// TIA Portal V17 export
// export: Created 2024-09-03T21:54:53.6894655Z, ExportSetting WithDefaults, DisplayName Totally Integrated Automation Portal, DisplayVersion V17 Update 7, DisplayName TIA Portal Openness, DisplayVersion V17 Update 7, DisplayName TIA Portal Version Control Interface, DisplayVersion V17, DisplayName SINAMICS Startdrive Advanced, DisplayVersion V17 SP2, DisplayName SINAMICS Startdrive G110M, G120, G120C, G120D, G120P, G115D, DisplayVersion V17 SP2, DisplayName SINAMICS Startdrive G130, G150, S120, S150, SINAMICS MV, S210, DisplayVersion V17 SP2, DisplayName STEP 7 Professional, DisplayVersion V17 Update 7, DisplayName STEP 7 Safety, DisplayVersion V17 Update 6, DisplayName WinCC Advanced / Unified PC, DisplayVersion V17 Update 7
ORGANIZATION_BLOCK "Startup"   // OB124, LAD, Startup
TITLE = "Complete Restart"
{ S7_Optimized_Access := 'TRUE' }
VERSION : 0.1
// stored: AutoNumber true, IsIECCheckEnabled false, SetENOAutomatically false
   VAR_INPUT
      LostRetentive : Bool;   // True if retentive data are lost
      LostRTC : Bool;   // True if date and time are lost
   END_VAR
BEGIN

REGION Network 1: Braketest or mastering requred
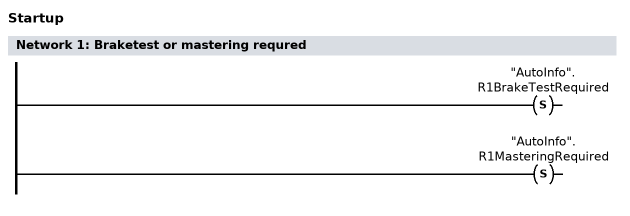
   RUNG wire#powerrail
      S_Coil( "AutoInfo".R1BrakeTestRequired )
   END_RUNG
   RUNG wire#powerrail
      S_Coil( "AutoInfo".R1MasteringRequired )
   END_RUNG
   // the same network as SCL:
   "AutoInfo".R1BrakeTestRequired := TRUE;
   "AutoInfo".R1MasteringRequired := TRUE;
END_REGION

REGION Network 2 (SCL)
       "DevicesData"."TA1-3MA".OverAcc := "StationParameters".Servo.OverAcc;
       "DevicesData"."TA1-3MA".OverDec := "StationParameters".Servo.OverDec;
       "DevicesData"."TA1-3MA".OverV := "StationParameters".Servo.OverV;
       "DevicesData"."TA1-3MA".Velocity := "StationParameters".Servo.Velocity;
END_REGION

REGION Network 3 (SCL)
   "setup_DB".minL := 100.0;
   "setup_DB".minR := "setup_DB".minL;
END_REGION
END_ORGANIZATION_BLOCK
